                   (* Call MC_Command*)
                    instGearInPos(Master := master,
                                  Slave := axis,
                                  Enable := statBasicCommand.8 OR statFirstCycleBasicMotion,(* Input: gearInAbsolute*)
                                  GearRatio := statRatioNumerator,
                                  (*RatioDenominator :=  statRatioDenominator,*)
                                  (*MasterSyncPosition :=  statMasterSyncPosition,*)
                                  (*SlaveSyncPosition :=  statSlaveSyncPosition,*)
                                  (*SyncProfileReference :=  statSyncProfileReference,*)
                                  (*MasterStartDistance :=  statMasterStartDistance,*)

                                  Acceleration :=  statAcceleration,
                                  Deceleration :=  statDeceleration,
                                  Jerk := statJerk,
                    (*SyncDirection :=  statSyncDirection*) );


                   (* Evaluate MC_Command*)
                    IF (instGearInPos.Busy = FALSE) AND
                        (instGearInPos.Error = FALSE) AND
                        (instGearInPos.CommandAborted = FALSE) AND
                    (*( instGearInPos.StartSync = FALSE) AND*)
                        (instGearInPos.InGear = FALSE)
                        THEN
                       (* Return to NO_SELECTION if command finished*)
                        statBasicMotionState := NO_SELECTION;

                    ELSIF (instGearInPos.Error = TRUE) THEN
                       (* Errorhandling*)
                        statStatus                    := ERR_MC_GEARINPOS;
                        statErrorAutoCleared          := TRUE;
                        diagnostics                   := statDiagnostics;
                        diagnostics.subfunctionStatus := instGearInPos.ErrorId;
                        statRatioChangeOnTheFly       := FALSE;
                       (* Set next state*)
                        statFBState          := AXIS_STOP_ON_ERROR_SELECTION;
                        statBasicMotionState := NO_SELECTION;

                    ELSE
                        ;(* Command selected*)
                    END_IF;

                   (* Write MC_Command outputs to internal variable*)
                    statExeOfBasicMotion   := 16#0;
                    statExeOfBasicMotion.0 := instGearInPos.Busy;
                    statExeOfBasicMotion.2 := instGearInPos.CommandAborted;
                    statExeOfBasicMotion.3 := instGearInPos.Error;
                    (*statExeOfBasicMotion.6 :=  instGearInPos.StartSync;*)
                    (*statExeOfBasicMotion.6 :=  instGearInPos.StartSync;*)
                    statExeOfBasicMotion.7 := instGearInPos.InGear;
                {END_REGION}

                CAM_IN_SELECTED:
                   (* Additional feature (applicative): Check DB of Cam *)
                    {REGION "CAM_IN_SELECTED"}
                   (* Firstcycle of command*)
                    IF (statFirstCycleBasicMotion = TRUE) THEN
                        (*IF TypeOfDB( cam) = TO_Cam*)
                        IF tempFalse = FALSE
                            THEN
                            (*statCam :=  cam;*)
                           (* Reset CAM_IN command *)
(*                            instCamIn(Master := master,
                                      Slave := axis,
                                      (*Cam :=  statCam,*)
                                      Execute := FALSE);
*)
                            statApplicativeBasicMotionError := FALSE;
                            statApplicationMode             := configuration.camIn.applicationMode;
                        ELSE
                           (* Errorhandling - Invalid cam*)
                            statStatus                      := ERR_INVALID_CAM;
                            statErrorAutoCleared            := TRUE;
                            diagnostics.subfunctionStatus   := 0;
                            diagnostics                     := statDiagnostics;
                            statApplicativeBasicMotionError := TRUE;
                           (* Set next state*)
                            statFBState          := AXIS_STOP_ON_ERROR_SELECTION;
                            statBasicMotionState := NO_SELECTION;
                        END_IF;
                    END_IF;

                    IF (statApplicativeBasicMotionError = FALSE) THEN

                       (* Write MC Parameters*)
(*                        instCamIn.CamTableID                 := configuration.camIn.tableID;
                        instCamIn.StartMode                  := configuration.camIn.startMode;
                        instCamIn.MasterOffset               := configuration.camIn.masterOffset;
                        instCamIn.SlaveOffset                := configuration.camIn.slaveOffset;
                        instCamIn.MasterScaling              := configuration.camIn.masterScaling;
                        instCamIn.SlaveScaling               := configuration.camIn.slaveScaling;
						instCamIn.StartMode     			 := configuration.camIn.startMode;
                        instCamIn.Options.ActivationMode     := configuration.camIn.ActivationMode;
                        instCamIn.Options.ActivationPosition := configuration.camIn.ActivationPosition;
*)
                       (* Call MC_Command*)
(*                        instCamIn(Master := master,
                                  Slave := axis,
*)  //                                Execute := statBasicCommand.9 OR statFirstCycleBasicMotion);
(*
                       (* Evaluate MC_Command*)
                        IF ((instCamIn.Busy = FALSE) AND
                            (instCamIn.Error = FALSE) AND
                            (instCamIn.CommandAborted = FALSE) AND
                            (instCamIn.InSync = FALSE) AND
                        (*( instCamIn.StartSync = FALSE) AND*)
                            (statBasicCommand.9 = FALSE)
                            ) AND(* V1.0.2 Wait for one cycle EndOfProfile (--> Done) before function is finished at applicationMode ONCE*)
                            ((statApplicationMode <> APPLICATION_MODE_ONCE) OR
                            ((statApplicationMode = APPLICATION_MODE_ONCE) (*AND ( instCamIn.EndOfProfile = FALSE)*) ))
                            THEN
                           (* Return to NO_SELECTION if command finished*)
                            statBasicMotionState := NO_SELECTION;

                        ELSIF (instCamIn.Error = TRUE) THEN
                           (* Errorhandling*)
                            statStatus                    := ERR_MC_CAMIN;
                            statErrorAutoCleared          := TRUE;
                            diagnostics.subfunctionStatus := instCamIn.ErrorId;
                            diagnostics.basicMotionState  := statBasicMotionState;
                            statFBState                   := AXIS_STOP_ON_ERROR_SELECTION;
                            statBasicMotionState          := NO_SELECTION;

                        ELSE
                            ;(* Command selected*)
                        END_IF;
*)
                       (* Write MC_Command outputs to internal variable*)
                        statExeOfBasicMotion   := 16#0;
//                        statExeOfBasicMotion.0 := instCamIn.Busy;
                        IF (statApplicationMode = APPLICATION_MODE_ONCE)
                            THEN
                            ; (*statExeOfBasicMotion.1 :=  instCamIn.EndOfProfile;*)
                        END_IF;

 //                       statExeOfBasicMotion.2 := instCamIn.CommandAborted;
 //                       statExeOfBasicMotion.3 := instCamIn.Error;
                        (*statExeOfBasicMotion.6 :=  instCamIn.StartSync;*)
//                        statExeOfBasicMotion.7 := instCamIn.InSync;

                    ELSE
                        ;(* InValid cam*)
                    END_IF;
            {END_REGION}

            ELSE
               (* Errorhandling*)
                statStatus                    := ERR_UNDEFINED_BASIC_MOTION_STATE;
                statErrorUserCleared          := TRUE;
                diagnostics                   := statDiagnostics;
                diagnostics.subfunctionStatus := 0;
               (* Set errorstate*)
                statFBState := FB_ERROR;
            END_CASE;

        RESET_GEARING:
           (* Abort waiting absolute gearing / camIn job if new basic motion job is selected (configuration.generalSettings.abortWaitingSyncCmd = TRUE)*)
            instGearIn(Master := master,
                       Slave := axis,
                       Execute := TRUE,
                       RatioNumerator := 1,
                       RatioDenominator := 1);(* Lowest possible gear ratio*)

            IF (instGearIn.InGear = TRUE) OR (instGearIn.CommandAborted = TRUE)
                THEN                                           (* Relative gearing command has aborted waiting absolute gearing job*)
                statMainSelectionState    := CALL_BASIC_MOTION;(* Execute new basic motion command*)
                tempStateChangeActive     := TRUE;
                statFirstCycleBasicMotion := TRUE;

            ELSIF (instGearIn.Error = TRUE)
                THEN
                statStatus                    := ERR_MC_GEARIN;
                diagnostics.subfunctionStatus := instGearIn.ErrorId;
               (*Errorhandling*)
                statErrorAutoCleared := TRUE;
                diagnostics          := statDiagnostics;
               (*Set next state*)
                statFBState            := AXIS_STOP_ON_ERROR_SELECTION;
                statMainSelectionState := CALL_BASIC_MOTION;
                statBasicMotionState   := NO_SELECTION;

            ELSE
                ;(* Command running*)
            END_IF;

           (* Write MC_Command outputs to internal variable*)
            statExeOfBasicMotion   := 16#0;
            statExeOfBasicMotion.0 := instGearIn.Busy;
    ELSE
       (* Errorhandling*)
        statStatus                    := ERR_UNDEFINED_MAIN_SELECTION_STATE;
        statErrorUserCleared          := TRUE;
        diagnostics                   := statDiagnostics;
        diagnostics.subfunctionStatus := 0;
       (* Set errorstate*)
        statFBState := FB_ERROR;
    END_CASE;

UNTIL (tempStateChangeActive = FALSE)
END_REPEAT;

{END_REGION}


(*----------------------------------------------------------------------------------------------*)
(*Execution of homing functionality *)
(*----------------------------------------------------------------------------------------------*)


{REGION "EXECUTION_OF_PASSIVE_HOMING"}
(*Statemachine for homing functionality*)
CASE statPassiveHomingState OF
   (* Selection of extended homing mode *) 
    NO_HOMING_ACTIVE:
        ;(* Do nothing*)

    STANDARD_HOMING:
       (* No additional features*)
        {REGION "STANDARD_HOMING"}
       (* Firstcycle of command*)
        IF (statFirstCycleHoming = TRUE) THEN
           (* Reset MC_HOME command*)
            instHome(Axis := axis,
                     bCalibrationCam := homingSensor,
                     Execute := FALSE);

            IF (statBasicMotionState = ACTIVE_HOMING_SELECTED) THEN
                statBasicMotionState := NO_SELECTION;
            END_IF;
        END_IF;

       (* Call MC_Command*)
        instHome(Axis := axis,
                 bCalibrationCam := homingSensor,
                 Execute := statExtendedCommand.2,(* Input: homing*)
                 Position := configuration.homing.position,
        (*Mode :=  configuration.homing.mode*) );

       (* Evaluate MC_Command*)
        IF (instHome.Busy = FALSE) AND
            (instHome.Done = FALSE) AND
            (instHome.CommandAborted = FALSE) AND
            (instHome.Error = FALSE)
            THEN
           (* Return to NO_SELECTION if command finished*)
            statPassiveHomingState := NO_HOMING_ACTIVE;

        ELSIF (instHome.Error = TRUE) THEN
           (* Errorhandling*)
            statStatus                    := ERR_MC_HOME;
            statErrorAutoCleared          := TRUE;
            diagnostics                   := statDiagnostics;
            diagnostics.subfunctionStatus := instHome.ErrorId;
            statPassiveHomingState        := NO_HOMING_ACTIVE;
           (* Set next state*)
            statFBState := AXIS_STOP_ON_ERROR_SELECTION;
        ELSE
            ;(* Command selected*)

        END_IF;

        statExeOfHoming   := 16#0;
        statExeOfHoming.0 := instHome.Busy;
        statExeOfHoming.1 := instHome.Done;
        statExeOfHoming.2 := instHome.CommandAborted;
        statExeOfHoming.3 := instHome.Error;
{END_REGION}

ELSE
   (* Errorhandling*)
    statStatus                              := ERR_INVALID_HOMING_EXTENDED_MODE;
    statErrorAutoCleared                    := TRUE;
    diagnostics                             := statDiagnostics;
    diagnostics.subfunctionStatus           := 0;
    statDiagnostics.basicMotionState        := statBasicMotionState;
    statDiagnostics.superimposedMotionState := statSupImpMotionState;
   (* Set next state*)
    statFBState            := AXIS_STOP_ON_ERROR_SELECTION;
    statBasicMotionState   := NO_SELECTION;
    statPassiveHomingState := NO_HOMING_ACTIVE;
END_CASE;

{END_REGION}


(*----------------------------------------------------------------------------------------------*)
(*Execution of functionalities of superimposed coordinate system*)
(*----------------------------------------------------------------------------------------------*)


{REGION "EXECUTION_OF_SUPERIMPOSED_COMMANDS"}
(*Statemachine for superimposed motion commands*)
(*Write diagnostics*)

statDiagnostics.basicMotionState        := statBasicMotionState;
statDiagnostics.superimposedMotionState := statSupImpMotionState;

CASE statSupImpMotionState OF
    NO_SELECTION:
        ;(* Do nothing*)

    POS_SUPERIMPOSED_SELECTED:
       (* Additional features (applicative) : Specified direction*)
        {REGION "POS_SUPERIMPOSED_SELECTED;"}
       (* Firstcycle of command*)
        IF (statFirstCycleSupImpMotion = TRUE) THEN
           (* Configurate the direction of rotation*)
            IF ((configuration.posSuperimposed.direction = 0) AND (configuration.posSuperimposed.distance >= 0.0))(* Sign of distance is evaluated*)
                OR
                (configuration.posSuperimposed.direction = FORWARD_DIR)(* Positive direction*)
                THEN
                statSupImpMotionPosition := ABS(configuration.posSuperimposed.distance);
               (* Reset MC_MOVESUPERIMPOSED command*)
                instMoveSuperimposed(Axis := axis,
                                     Execute := FALSE);

                statApplicativeSupImpMotionError := FALSE;
            ELSIF ((configuration.posSuperimposed.direction = 0) AND (configuration.posSuperimposed.distance < 0.0))(* Sign of distance is evaluated*)
                OR
                (configuration.posSuperimposed.direction = BACKWARD_DIR)(* Negative direction *)
                THEN
                statSupImpMotionPosition := -ABS(configuration.posSuperimposed.distance);
               (* Reset MC_MOVESUPERIMPOSED command*)
                instMoveSuperimposed(Axis := axis,
                                     Execute := FALSE);

                statApplicativeSupImpMotionError := FALSE;

            ELSE
               (* Errorhandling - Invalid direction*)
                statStatus                       := ERR_INVALID_POS_SUPERIMPOSED_DIR;
                statErrorAutoCleared             := TRUE;
                diagnostics                      := statDiagnostics;
                diagnostics.subfunctionStatus    := 0;
                statApplicativeSupImpMotionError := TRUE;
               (* Set next state*)
                statFBState           := AXIS_STOP_ON_ERROR_SELECTION;
                statSupImpMotionState := NO_SELECTION;
            END_IF;
        END_IF;

        IF (statApplicativeSupImpMotionError = FALSE) THEN
           (* Call MC_Command*)
            instMoveSuperimposed(Axis := axis,
                                 Execute := statSupImpCommand.0,(* Input: posSuperimposed*)
                                 Distance := statSupImpMotionPosition,
                                 VelocityDiff := configuration.posSuperimposed.velocityDiff,
                                 Acceleration := configuration.posSuperimposed.acceleration,
                                 Deceleration := configuration.posSuperimposed.deceleration,
                                 Jerk := configuration.posSuperimposed.jerk);

           (* Evaluate MC_Command*)
            IF (instMoveSuperimposed.Busy = FALSE) AND
                (instMoveSuperimposed.Error = FALSE) AND
                (instMoveSuperimposed.Done = FALSE) AND
                (instMoveSuperimposed.CommandAborted = FALSE)
                THEN
               (* Return to NO_SELECTION if command finished*)
                statSupImpMotionState := NO_SELECTION;

            ELSIF (instMoveSuperimposed.Error = TRUE) THEN
               (* Errorhandling*)
                statStatus                    := ERR_MC_MOVESUPERIMPOSED;
                statErrorAutoCleared          := TRUE;
                diagnostics                   := statDiagnostics;
                diagnostics.subfunctionStatus := instMoveSuperimposed.ErrorId;
               (* Set next state*)
                statFBState           := AXIS_STOP_ON_ERROR_SELECTION;
                statSupImpMotionState := NO_SELECTION;

            ELSE
                ;(* command selected*)
            END_IF;

            statExeOfSupImpMotionState   := 16#0;
            statExeOfSupImpMotionState.0 := instMoveSuperimposed.Busy;
            statExeOfSupImpMotionState.1 := instMoveSuperimposed.Done;
            statExeOfSupImpMotionState.2 := instMoveSuperimposed.CommandAborted;
            statExeOfSupImpMotionState.3 := instMoveSuperimposed.Error;
        END_IF;
    {END_REGION}

    PHASING_SELECTED:
       (* Additional features (applicative) : Change setpoint on the fly (phaseShift)*)
        {REGION "PHASING_SELECTED"}
       (* Firstcycle of command*)
        IF (statFirstCycleSupImpMotion = TRUE) THEN
           (* Reset MC_PHASING_ABSOLUTE command*)
            instPhasingAbsolute(Master := master,
                                Slave := axis,
                                Execute := FALSE);

           (* Reset MC_PHASING_RELATIVE command*)
            instPhasingRelative(Master := master,
                                Slave := axis,
                                Execute := FALSE);

            statPhaseShift               := configuration.phasing.phaseShift;
            statVelocity                 := configuration.phasing.velocity;
            statAcceleration             := configuration.phasing.acceleration;
            statDeceleration             := configuration.phasing.deceleration;
            statJerk                     := configuration.phasing.jerk;
            statPhaseAbsolute            := configuration.phasing.phaseAbsolute;
            statChangePhaseShiftOnTheFly := configuration.phasing.phaseShiftChangeOnTheFly;

        ELSIF ((statChangePhaseShiftOnTheFly = TRUE) AND
            (configuration.phasing.phaseShift <> statPhaseShift)) AND
            (statPhaseAbsolute = TRUE) AND
            (instPhasingAbsolute.CommandAborted = FALSE)
            THEN
           (* Reset MC_PHASING_ABSOLUTE command - Phaseshift on the fly is only possible at phasing absolut*)
            instPhasingAbsolute(Master := master,
                                Slave := axis,
                                Execute := FALSE);

            statPhaseShift := configuration.phasing.phaseShift;
        END_IF;

       (* Select phasing absolut or relative *)
        IF (statPhaseAbsolute = TRUE) THEN
           (* Absolute phasing*)
           (* Call MC_Command*)
            instPhasingAbsolute(Master := master,
                                Slave := axis,
                                Execute := statSupImpCommand.1,(* Input: phasing*)
                                PhaseShift := statPhaseShift,
                                Velocity := statVelocity,
                                Acceleration := statAcceleration,
                                Deceleration := statDeceleration,
                                Jerk := statJerk);

           (* Evaluate MC_Command*)
            IF (instPhasingAbsolute.Busy = FALSE) AND
                (instPhasingAbsolute.Error = FALSE) AND
                (instPhasingAbsolute.Done = FALSE) AND
                (instPhasingAbsolute.CommandAborted = FALSE)
                THEN
               (* Return to NO_SELECTION if command finished*)
                statSupImpMotionState := NO_SELECTION;

            ELSIF (instPhasingAbsolute.Error = TRUE) THEN
               (* Errorhandling*)
                statStatus                    := ERR_MC_PHASINGABSOLUTE;
                statErrorAutoCleared          := TRUE;
                diagnostics                   := statDiagnostics;
                diagnostics.subfunctionStatus := instPhasingAbsolute.ErrorId;
                statChangePhaseShiftOnTheFly  := FALSE;
               (* Set next state*)
                statFBState           := AXIS_STOP_ON_ERROR_SELECTION;
                statSupImpMotionState := NO_SELECTION;

            ELSE
                ;(* Command busy*)
            END_IF;

            statExeOfSupImpMotionState   := 16#0;
            statExeOfSupImpMotionState.0 := instPhasingAbsolute.Busy;
            statExeOfSupImpMotionState.1 := instPhasingAbsolute.Done;
            statExeOfSupImpMotionState.2 := instPhasingAbsolute.CommandAborted;
            statExeOfSupImpMotionState.3 := instPhasingAbsolute.Error;

        ELSE
           (* Relative phasing  *)
           (* Call MC_Command*)
            instPhasingRelative(Master := master,
                                Slave := axis,
                                Execute := statSupImpCommand.1,(* Input: phasing*)
                                PhaseShift := statPhaseShift,
                                Velocity := statVelocity,
                                Acceleration := statAcceleration,
                                Deceleration := statDeceleration,
                                Jerk := statJerk);

           (* Evaluate MC_Command*)
            IF (instPhasingRelative.Busy = FALSE) AND
                (instPhasingRelative.Error = FALSE) AND
                (instPhasingRelative.Done = FALSE) AND
                (instPhasingRelative.CommandAborted = FALSE)
                THEN
               (* Return to NO_SELECTION if command finished*)
                statSupImpMotionState := NO_SELECTION;

            ELSIF (instPhasingRelative.Error = TRUE) THEN
               (* Errorhandling*)
                statStatus                    := ERR_MC_PHASINGRELATIVE;
                statErrorAutoCleared          := TRUE;
                diagnostics                   := statDiagnostics;
                diagnostics.subfunctionStatus := instPhasingRelative.ErrorId;
                statChangePhaseShiftOnTheFly  := FALSE;
               (* Set next state*)
                statFBState           := AXIS_STOP_ON_ERROR_SELECTION;
                statSupImpMotionState := NO_SELECTION;
            ELSE
                ;(* Command selected*)
            END_IF;

            statExeOfSupImpMotionState   := 16#0;
            statExeOfSupImpMotionState.0 := instPhasingRelative.Busy;
            statExeOfSupImpMotionState.1 := instPhasingRelative.Done;
            statExeOfSupImpMotionState.2 := instPhasingRelative.CommandAborted;
            statExeOfSupImpMotionState.3 := instPhasingRelative.Error;
        END_IF;
{END_REGION}

ELSE
   (* Errorhandling*)
    statStatus                    := ERR_UNDEFINED_SUPERIMPOSED_MOTION_STATE;
    statErrorUserCleared          := TRUE;
    diagnostics                   := statDiagnostics;
    diagnostics.subfunctionStatus := 0;
   (* Set errorstate*)
    statFBState := FB_ERROR;
END_CASE;

{END_REGION}

(*----------------------------------------------------------------------------------------------*)
(*Execution of torquelimiting functionality*)
(*----------------------------------------------------------------------------------------------*)


{REGION "EXECUTION_OF_TORQUELIMTING"}
(*Statemachine for torquelimiting *)
REPEAT
    tempStateChangeActive := FALSE;
    CASE statTorqueLimitingState OF
        NO_TORQUE_LIMITING_ACTIVE:
            ;(* Torquelimiting disable*)
       (*  instTorqueLimiting(Axis :=  axis, V01.00.03 Dont Call MC_TORQUELIMITING if disabled*)
       (*                     Enable := FALSE);*)

        TORQUE_LIMITING_DISABLE:
           (* Torquelimiting disable*)
            instTorqueLimiting(Axis := axis,
                               Enable := FALSE);

           (* Check state of torque limting*)
            IF (instTorqueLimiting.Busy = FALSE)
                THEN
               (* set next state*)
                statTorqueLimitingState := NO_TORQUE_LIMITING_ACTIVE;
            ELSE
                ;(* Waiting for MC_Torquelimiting is not busy*)
            END_IF;

        TORQUE_LIMTING_SELECTED:
           (* No extended homing function active*)
            instTorqueLimiting(Axis := axis,
                               Enable := statExtendedCommand.1,
                               TLimit := configuration.torqueLimiting.TorqueLimit,
                               Mode := configuration.torqueLimiting.mode);

            IF (instTorqueLimiting.Busy = FALSE) THEN
               (* Reset state*)
                statTorqueLimitingState := NO_TORQUE_LIMITING_ACTIVE;
            END_IF;

        (*
	        V1.00.03 Not required anymore
	       AUTOMATIC_MODE_CHANGE:
	        // In this state the torquelimiting function is operating with Mode 1 (Fixed stop detection) until inClamping = FALSE
	         instTorqueLimiting(Axis :=  axis,
	                            Enable := TRUE,
	                            Limit :=  configuration.homing.extendedModeTorqueLimit); // V01.00.03 Always use configured value
	        
	        IF ( configuration.torqueLimiting.mode =  MODE_FIXED_STOP_DETECTION)
	          OR ( instTorqueLimiting.InClamping = FALSE)
	        THEN
	          // Change state
	           statTorqueLimitingState :=  TORQUE_LIMTING_SELECTED;
	           tempStateChangeActive := TRUE;
	        ELSE
	          ; // Wait for InClamping = FALSE
	        END_IF;
	        *)

        FIXED_STOP_DETECTION_ACTIVE:
           (* Extended homing function active*)
            instTorqueLimiting(Axis := axis,
                               Enable := TRUE,
                               TLimit := configuration.homing.extendedModeTorqueLimit,(* V01.00.03 Always use configured value*)
                               Mode := MODE_FIXED_STOP_DETECTION);

            IF ((statHomingSubState = HOMING_IDLE) AND (statBasicMotionState = ACTIVE_HOMING_SELECTED))
                THEN
               (* Fixed stop process has finished - Axis is still in clamping*)
                statTorqueLimitingState := FIXED_STOP_DETECTION_FINISHED;
                tempStateChangeActive   := TRUE;

            ELSIF (statBasicMotionState <> ACTIVE_HOMING_SELECTED)
                THEN
               (* Error occurred - change state depending on inClamping*)
                IF (instTorqueLimiting.InClamping = TRUE)
                    THEN
                   (* Axis is in clamping*)
                    statTorqueLimitingState := FIXED_STOP_DETECTION_ERROR_IN_CLAMPING;
                    tempStateChangeActive   := TRUE;
                ELSE
                   (* Axis is in not clamping*)
                    statTorqueLimitingState := FIXED_STOP_DETECTION_ERROR_NOT_IN_CLAMPING;
                    tempStateChangeActive   := TRUE;
                END_IF;

            ELSE
                ;(* Fixed stop detection is running*)
            END_IF;

        FIXED_STOP_DETECTION_FINISHED:
           (* Homing on fixed stop process has finished*)
            instTorqueLimiting(Axis := axis,
                               Enable := TRUE,
                               TLimit := configuration.homing.extendedModeTorqueLimit,(* V01.00.03 Always use configured value*)
                               Mode := MODE_FIXED_STOP_DETECTION);

            IF (instTorqueLimiting.InClamping = FALSE)
                THEN
               (* InClamping = FALSE*)
                IF (statExtendedCommand.1 = TRUE)(* Torquelimiting*)
                    THEN
                    statTorqueLimitingState := TORQUE_LIMTING_SELECTED;
                ELSE
                    statTorqueLimitingState := TORQUE_LIMITING_DISABLE;
                END_IF;

                tempStateChangeActive := TRUE;
            ELSE
               (* InClamping = TRUE*)
                IF (statExtendedCommand.1 = TRUE)(* Torquelimiting*)
                    AND
                    (configuration.torqueLimiting.mode = MODE_FIXED_STOP_DETECTION)
                    THEN
                   (* Change State*)
                    statTorqueLimitingState := TORQUE_LIMTING_SELECTED;
                    tempStateChangeActive   := TRUE;
                ELSE
                    ;(* Wait for inClamping = FALSE*)
                END_IF;
            END_IF;

        FIXED_STOP_DETECTION_ERROR_IN_CLAMPING:
           (* Errorstate, torquelimiting is still active and axis not in clamping*)
            instTorqueLimiting(Axis := axis,
                               Enable := TRUE,
                               TLimit := configuration.homing.extendedModeTorqueLimit,(* V01.00.03 Always use configured value*)
                               Mode := MODE_FIXED_STOP_DETECTION);

            IF (instTorqueLimiting.InClamping = FALSE)
                THEN
               (* InClamping = FALSE -> reset torque limiting state*)
                statTorqueLimitingState := TORQUE_LIMITING_DISABLE;
               (* Torquelimiting disable*)
                tempStateChangeActive := TRUE;
            END_IF;

        FIXED_STOP_DETECTION_ERROR_NOT_IN_CLAMPING:
           (* Errorstate, torquelimiting is still active and axis in clamping*)
            instTorqueLimiting(Axis := axis,
                               Enable := TRUE,
                               TLimit := configuration.homing.extendedModeTorqueLimit,(* V01.00.03 Always use configured value*)
                               Mode := MODE_FIXED_STOP_DETECTION);

            IF (instTorqueLimiting.InClamping = TRUE)
                THEN
               (* InClamping = TRUE -> change state*)
                statTorqueLimitingState := FIXED_STOP_DETECTION_ERROR_IN_CLAMPING;
                tempStateChangeActive   := TRUE;

            ELSIF (statBasicMotionState <> NO_SELECTION) OR (statSupImpMotionState <> NO_SELECTION) OR (statPassiveHomingState <> NO_HOMING_ACTIVE)
                THEN
               (* New valid command is set -> reset error state*)
                statTorqueLimitingState := TORQUE_LIMITING_DISABLE;
                tempStateChangeActive   := TRUE;

            ELSE
                ;(* Waiting for new command or axis is getting in clamping*)
            END_IF;
    ELSE
       (* Errorhandling*)
        statStatus                          := ERR_UNDEFINED_TORQUE_LIMITING_STATE;
        statErrorUserCleared                := TRUE;
        diagnostics.basicMotionState        := statBasicMotionState;
        diagnostics.superimposedMotionState := statSupImpMotionState;
        diagnostics.subfunctionStatus       := 0;
       (* Set errorstate*)
        statFBState := FB_ERROR;
    END_CASE;
UNTIL (tempStateChangeActive = FALSE)
END_REPEAT;

(* Evaluate MC_Command*)
IF (instTorqueLimiting.Error = TRUE) AND ((statTorqueLimitingErrorOld = FALSE) OR (statStatus = STATUS_SUBSEQUENT_CALL)) THEN
   (* Errorhandling*)
    statStatus                          := ERR_MC_TORQUELIMITING;
    statErrorAutoCleared                := TRUE;
    diagnostics.basicMotionState        := statBasicMotionState;
    diagnostics.superimposedMotionState := statSupImpMotionState;
    diagnostics.subfunctionStatus       := instTorqueLimiting.ErrorId;
    statFBState                         := AXIS_STOP_ON_ERROR_SELECTION;

ELSIF (instTorqueLimiting.Error = FALSE) AND ((statTorqueLimitingErrorOld = TRUE) AND (statStatus = ERR_MC_TORQUELIMITING)) THEN
    statStatus           := STATUS_SUBSEQUENT_CALL;
    statErrorAutoCleared := FALSE;
ELSE
    ;
END_IF;

statTorqueLimitingErrorOld := instTorqueLimiting.Error;
{END_REGION}


(*----------------------------------------------------------------------------------------------*)
(* Selection of StopOnError / implementation of fastStop*)
(*----------------------------------------------------------------------------------------------*)

{REGION "STOP_ON_ERROR"}

(*Check for stopping if error occurred during execution of motion commands*)

IF (statFBState = AXIS_STOP_ON_ERROR_SELECTION)
    THEN
    statBasicMotionState   := NO_SELECTION;
    statSupImpMotionState  := NO_SELECTION;
    statPassiveHomingState := NO_HOMING_ACTIVE;

    IF (configuration.generalSettings.stopOnError = TRUE)
        THEN
       (* Read Statusword only when not already read out*)
        IF (tempStatusWord = 16#0)
            THEN
            tempStatusWord := axis.NcToPlc.StateDWord;
        END_IF;

       (* Evaluate error*)
        IF tempStatusWord.0 THEN
            ;(* Axis enabled*)
            IF (tempStatusWord.1 = TRUE) THEN
                ;(* TO Alarm present*)
                statFBState := AXIS_MOTION;
            ELSE
               (* No TO alarm present, set fastStop*)
                statBasicMotionState      := FAST_STOP_SELECTED;
                statFirstCycleBasicMotion := TRUE;
                statFBState               := AXIS_STOP_ON_ERROR_EXECUTION;
            END_IF;

        ELSE
            ;(* Axis disabled*)
            statFBState := AXIS_MOTION;
        END_IF;

    ELSE
       (* Dont StopOnError*)
        statFBState := AXIS_MOTION;
    END_IF;
END_IF;

(*Implementation of fastStop*)
IF (statBasicMotionState = FAST_STOP_SELECTED) THEN
   (* Additional feature: Load emergency stop dynamics (TO) if no valid dynamics are configured for fastStop*)
    {REGION "FASTSTOP SELECTED"}
   (* Firstcycle of command*)
    IF (statFirstCycleBasicMotion = TRUE) THEN
       (* Reset HALT command*)
        instHalt(Axis := axis,
                 Execute := FALSE);

        statFirstCycleDone := TRUE;
       (* Check dynamics for fastStop*)
       (* Load TO emergency Stop dynamics if value <=0 for deceleration is configured*)
        IF (configuration.fastStop.deceleration <= 0)(* V1.0.2 Read TO emergencyStop deceleration only IF fastStop.deceleration <= 0*)
            THEN
           (* Invalid fastStop dynamics configured - read emergency stop dynamics from TO*)
            (*statDeceleration :=  axis.DynamicDefaults.EmergencyDeceleration;*)
            statDeceleration := configuration.fastStop.deceleration;
        ELSE
           (* Valid fastStop dynamics configured*)
            statDeceleration := configuration.fastStop.deceleration;
        END_IF;

        statJerk              := configuration.fastStop.jerk;             (* V1.0.2 Use always configuration for jerk value*)
        statAbortAcceleration := configuration.fastStop.abortAcceleration;(* V1.0.2 Use always configuration*)
    END_IF;

   (* Call of MC_Command*)
    instHalt(Axis := axis,
             Execute := (statBasicCommand.0 OR statFirstCycleBasicMotion),
             Deceleration := statDeceleration,
             (*AbortAcceleration :=  statAbortAcceleration,*)
             Jerk := statJerk);

   (* Evaluate MC_Command*)
    IF (instHalt.Busy = FALSE) AND
        (instHalt.Error = FALSE) AND
        (instHalt.Done = FALSE) AND
        (instHalt.CommandAborted = FALSE)
        THEN
       (* Return to NO_SELECTION if command finished*)
        statFBState          := AXIS_MOTION;
        statBasicMotionState := NO_SELECTION;

    ELSIF (instHalt.Done = TRUE)
        THEN
        IF (statFirstCycleDone = TRUE)
            THEN
           (* Command is reset*)
            IF (instTorqueLimiting.Error = FALSE)(* V1.00.03 Dont reset error is pending*)
                THEN
               (* Reset status not if torquelimiting error is pending*)
                statStatus           := STATUS_SUBSEQUENT_CALL;
                statErrorAutoCleared := FALSE;
            END_IF;

            statFirstCycleDone := FALSE;
        END_IF;

    ELSIF (instHalt.Error = TRUE)
        THEN
       (* Errorhandling*)
        statStatus                          := ERR_MC_HALT;
        statErrorAutoCleared                := TRUE;
        diagnostics                         := statDiagnostics;
        diagnostics.basicMotionState        := statBasicMotionState;
        diagnostics.superimposedMotionState := statSupImpMotionState;
        diagnostics.subfunctionStatus       := instHalt.ErrorId;

    ELSE
        ;(* Command selected*)
    END_IF;

   (* Write MC_Command outputs to internal variable*)
    statExeOfBasicMotion   := 0;
    statExeOfBasicMotion.0 := instHalt.Busy;
    statExeOfBasicMotion.1 := instHalt.Done;
    statExeOfBasicMotion.2 := instHalt.CommandAborted;
    statExeOfBasicMotion.3 := instHalt.Error;
    {END_REGION}
END_IF;

{END_REGION}

(*----------------------------------------------------------------------------------------------*)
(*Store values and reset variables										*)
(*----------------------------------------------------------------------------------------------*)

{REGION "STORE_AND_RESET"}
(*Reset variables to determine first cycle of a new command*)
IF (statFirstCycleReset = TRUE) THEN
    statFirstCycleReset := FALSE;
END_IF;

IF (statFirstCycleHoming = TRUE) THEN
    statFirstCycleHoming := FALSE;
END_IF;

statHomingOld := tempHoming;

IF (statFirstCycleBasicMotion = TRUE) THEN
    statFirstCycleBasicMotion := FALSE;
END_IF;

statBasicCommandOld := statBasicCommand;

IF (statFirstCycleSupImpMotion = TRUE) THEN
    statFirstCycleSupImpMotion := FALSE;
END_IF;

statSupImpCommandOld := statSupImpCommand;

(*Store last values for edge detection*)
statEnableOld          := enable;
statEnableAxisOld      := enableAxis;
statExtendedCommandOld := statExtendedCommand;
statPowerErrorOld      := instPower.Error;
{END_REGION}


(*----------------------------------------------------------------------------------------------*)
(*Writing outputs													*)
(*----------------------------------------------------------------------------------------------*)

{REGION "WRITING_OF_OUTPUTS"}
(*Writing status outputs*)
resetActive := (statResetState = CMD_BUSY);

IF (statErrorUserCleared = TRUE) THEN
    ;(* Reset variables at ErrorUserCleared*)
    statBasicMotionState       := NO_SELECTION;
    statExeOfBasicMotion       := NO_SELECTION;
    statSupImpMotionState      := NO_SELECTION;
    statExeOfSupImpMotionState := NO_SELECTION;
    statExeOfHoming            := NO_SELECTION;
END_IF;

IF (instPower.Status = TRUE)
    THEN
   (* Axis enabled*)
    axisEnabled := TRUE;

ELSIF (instPower.Error = TRUE) AND (instPower.Status = FALSE)
    THEN
   (* Reset status if error occurred*)
    axisEnabled := FALSE;

ELSIF (instPower.Busy = FALSE)
    THEN
   (* Reset if MC_Power is not busy*)
    axisEnabled := FALSE;
ELSE
    ;
END_IF;

{REGION "WRITING_BASICMOTION_OUTPUTS"}
(*Writing Busy, Done and Aborted outputs for basic motion commands*)
IF (statBasicMotionState > NO_SELECTION) AND (statBasicMotionState < ACTIVE_HOMING_SELECTED)
    THEN
    commandBusy    := statExeOfBasicMotion.0;
    commandDone    := statExeOfBasicMotion.1;
    commandAborted := statExeOfBasicMotion.2;
    inVelocity     := statExeOfBasicMotion.4;
    inSync         := statExeOfBasicMotion.7;
    startSync      := statExeOfBasicMotion.6;
ELSE
    commandBusy    := FALSE;
    commandDone    := FALSE;
    commandAborted := FALSE;
    inVelocity     := FALSE;
    inSync         := FALSE;
    startSync      := FALSE;
END_IF;

(*Writing outputs up to LAxisCtrl_SpeedAxis*)
IF (statTorqueLimitingState = TORQUE_LIMTING_SELECTED)
(*OR ( statTorqueLimitingState =  AUTOMATIC_MODE_CHANGE) V1.0.3 TorqueLimtinig = TRUE, only when respective value used *)
    THEN
    torqueLimitingSelected := TRUE;
ELSE
    torqueLimitingSelected := FALSE;
END_IF;

inLimitation         := instTorqueLimiting.InLimitation;
fastStopSelected     := statBasicMotionState.0;
stopSelected         := statBasicMotionState.1;
jogSelected          := statBasicMotionState.2 OR statBasicMotionState.3;
moveVelocitySelected := statBasicMotionState.4;
(* Writing outputs up to LAxisCtrl_PosAxis*)
inClamping          := instTorqueLimiting.InClamping;
posRelativeSelected := statBasicMotionState.5;
posAbsoluteSelected := statBasicMotionState.6;
(* Writing outputs up to LAxisCtrl_SyncAxisRelGearing*)
gearInRelativeSelected := statBasicMotionState.7;
(* Writing outputs up to LAxisCtrl_SyncAxisCamming*)
gearInAbsoluteSelected := statBasicMotionState.8;
camInSelected          := statBasicMotionState.9;
inSimulation           := instSyncMotionSimulation.InSimulation;
{END_REGION}
{REGION "WRITING_HOMING_OUTPUTS"}

(* Writing Busy, Done and Aborted outputs for homing*)
IF (statPassiveHomingState = STANDARD_HOMING)
    THEN
    homingSelected       := TRUE;
    homingCommandBusy    := statExeOfHoming.0;
    homingCommandDone    := statExeOfHoming.1;
    homingCommandAborted := statExeOfHoming.2;
ELSE
    IF (statBasicMotionState = ACTIVE_HOMING_SELECTED)
        THEN
        homingSelected       := TRUE;
        homingCommandBusy    := statExeOfBasicMotion.0;
        homingCommandDone    := statExeOfBasicMotion.1;
        homingCommandAborted := statExeOfBasicMotion.2;
    ELSE
        homingSelected       := FALSE;
        homingCommandBusy    := FALSE;
        homingCommandDone    := FALSE;
        homingCommandAborted := FALSE;
    END_IF;
END_IF;

{END_REGION}
{REGION "WRITING_SUPERIMPOSED_OUTPUTS"}

(*Writing outputs for superimposed motion commands*)
IF (statSupImpMotionState <> NO_SELECTION)
    THEN
    superimposedBusy    := statExeOfSupImpMotionState.0;
    superimposedDone    := statExeOfSupImpMotionState.1;
    superimposedAborted := statExeOfSupImpMotionState.2;
ELSE
    superimposedBusy    := FALSE;
    superimposedDone    := FALSE;
    superimposedAborted := FALSE;
END_IF;

posSuperimposedSelected := statSupImpMotionState.0;
phasingSelected         := statSupImpMotionState.1;
{END_REGION}
{END_REGION}

(*----------------------------------------------------------------------------------------------*)
(*Error handling 													*)
(*----------------------------------------------------------------------------------------------*)

{REGION "ERROR_HANDLING"}
IF statErrorUserCleared THEN
    valid              := FALSE;
    busy               := TRUE;
    error              := TRUE;
    status             := statStatus;
    diagnostics.status := statStatus;

ELSIF statErrorAutoCleared THEN
    valid              := FALSE;
    busy               := TRUE;
    error              := TRUE;
    status             := statStatus;
    diagnostics.status := statStatus;

ELSE
   (* Process normal output values*)
    valid  := TRUE;
    error  := FALSE;
    status := statStatus;
END_IF;

{END_REGION}

(*Axis status function block call*)
(*instAxisStatus(stAxis := Axis.NcToPlc);*)

END_FUNCTION_BLOCK

// ---- Library/AxisControl/MC_TORQUELIMITING.TcPOU
FUNCTION_BLOCK MC_TORQUELIMITING
VAR_INPUT
	{attribute 'hide'} 
	Axis : AXIS_REF;
	Enable : BOOL;
	TLimit : LREAL;
	Mode : DINT;
END_VAR
VAR_OUTPUT
	InClamping : BOOL;
	InLimitation : BOOL;
	Busy : BOOL;
	Error : BOOL;
	ErrorId : WORD;
END_VAR
VAR
END_VAR

;

END_FUNCTION_BLOCK

// ---- Library/AxisControl/DataTypes/MC_SYNCHRONIZEDMOTIONSIMULATION.TcPOU
FUNCTION_BLOCK MC_SYNCHRONIZEDMOTIONSIMULATION

VAR_IN_OUT
	Slave	: AXIS_REF;	(* B *)
END_VAR


VAR_INPUT


	Enable : BOOL;

END_VAR
VAR_OUTPUT

	InSimulation	:BOOL;

Busy	:BOOL;

	Error	:BOOL;

ErrorId	:WORD;

END_VAR
VAR
END_VAR

;

END_FUNCTION_BLOCK

// ---- Library/Machine/Slitter/FunctionBlocks/FB_KnifeSharpening_old.TcPOU
FUNCTION_BLOCK FB_KnifeSharpening_old
VAR_INPUT

	machineRunning 				: BOOL;
	manualSharpening 			: BOOL;
	measuringWheelSensor 		: BOOL;
	knifeRunningMetersReset 		: BOOL;
	knifeEnabled 				: BOOL;
	measuringWheelDiameter 		: REAL	:= 154.2;
	sharpeningSetpoint 			: REAL	:= 100.0;
	sharpeningTime				: INT 		:= 5000;

END_VAR
VAR_OUTPUT

	sharpeningSolenoid 			: BOOL;
	knifeRunningMeters 			: INT;
	knifeRunningMetersTotal 		: DINT;


END_VAR
VAR

	measuringWheelSensorOld		: BOOL;

	instSharpeningTimeTON		: TON;
	manualSharpeningOld			: BOOL;
	knifeRunningMetersResetOld	: BOOL;

END_VAR

VAR PERSISTENT

	sensorPulseCounter1 			: DINT;	(*This variable increases every pulse of the measuring wheel and resets every time the knife is shapened*)
	sensorPulseCounter2 			: DINT;	(*This variable increases every pulse of the measuring wheel and resets manualy when the knife is replaced*)


END_VAR

VAR

END_VAR

VAR CONSTANT

	PI: REAL 					:= 3.14159265359;

END_VAR


(*==============================================================================================================================
CPNTeck - Automação industrial
(c)Copyright 2022 All Rights Reserved
_______________________________________________________________________________________________________________________________
Library: N/A 
Tested with: CX5140
Engineering: Twincat 2
Restrictions: -
Requirements: N/A
Functionality: This function block is used to sharp the knifes
Support: fabio@cpnteck.com.br
Note: Parameter comments are only available in language 'English (United States)'
_______________________________________________________________________________________________________________________________
Change log table:

Version  		| Date        			| Expert in charge  	| Changes applied
01.00.01		| 18.04.2023  		| Fabio Campion            | First released version



===============================================================================================================================*)


(*Measuring wheel pulse counter*)
IF measuringWheelSensor AND NOT measuringWheelSensorOld
AND knifeEnabled  THEN

	sensorPulseCounter1 := sensorPulseCounter1 + 1;
	sensorPulseCounter2 := sensorPulseCounter2 + 1;


END_IF

measuringWheelSensorOld := measuringWheelSensor;


(*Automatic / Manual shapening*)
IF knifeRunningMeters >= sharpeningSetpoint AND machineRunning
OR  manualSharpening AND NOT manualSharpeningOld  AND machineRunning THEN

	sensorPulseCounter1 := 0; (*Reset the measuring wheel pulse counter*)
	instSharpeningTimeTON.PT := DINT_TO_TIME(SharpeningTime); (*Set the timer setpoint*)
	instSharpeningTimeTON.IN := TRUE; (*Enable the timer*)
	sharpeningSolenoid := TRUE; (*Enable the sharpening solenoid*)

END_IF

ManualSharpeningOld := ManualSharpening;

IF instSharpeningTimeTON.Q  THEN

	sharpeningSolenoid := FALSE;
	instSharpeningTimeTON.IN := FALSE;

END_IF

IF knifeRunningMetersReset AND NOT knifeRunningMetersResetOld THEN

	sensorPulseCounter2 := 0;

END_IF

knifeRunningMetersResetOld := knifeRunningMetersReset;



(*Measuring wheel meters calculation*)
KnifeRunningMeters := TRUNC_INT((sensorPulseCounter1 * (MeasuringWheelDiameter * PI)) * 0.001);
KnifeRunningMetersTotal := TRUNC_INT((sensorPulseCounter2 * (MeasuringWheelDiameter * PI)) * 0.001);



instSharpeningTimeTON();

END_FUNCTION_BLOCK

// ---- Library/Machine/Slitter/FunctionBlocks/FB_PositionsGeneration.TcPOU
FUNCTION_BLOCK FB_PositionsGeneration
VAR_INPUT

	execute					: BOOL;	(*Execute function block*)
	machineConfig						: slitterConfig_TypeStruct;
	
END_VAR


VAR_IN_OUT

	currentOrder				: Order_TypeStruct;

END_VAR

VAR_OUTPUT

	error						: BOOL;
	done						: BOOL;
	busy						: BOOL;

END_VAR
VAR


	tempCurrentOrder				: Order_TypeStruct;

	executeOld 				: BOOL;
	firstOrderTotal 				: REAL;
	secondOrderTotal 			: REAL;
	firstKnifePosition 				: REAL;	(*First knife position*)
	topOrderIndex				: INT;		(*Top order index*)
	bottomOrderIndex			: INT;		(*Bottom order index*)
	toolPositionIndex 			: INT;		(*Tool position array index*)
	knifePositionTopIndex 			: INT ;	(*Knife position array index*)
	knifePositionBottomIndex 		: INT ;	(*Knife position array index*)
	scorerPositionTopIndex 		: INT ;	(*Knife position array index*)
	scorerPositionBottomIndex 		: INT ;	(*Knife position array index*)
	scorerPositionIndex			: INT;		(*Scorer position array index*)
	knifeEnabledIndex			: INT;		(*Knife enabled index*)
	scorerEnabledIndex			: INT;		(*Scorer enabled index*)
	knifeDistributionIndex			: INT;		(*Position distribution index*)
	scorerDistributionIndex			: INT;		(*Position distribution index*)
	toolPositionArrSize 			: INT ;	(*Tool position array size*)
	knifePositionArrSize 			: INT ;	(*Knife position array size*)
	scorerPositionArrSize 			: INT ;	(*Scorer position array size*)
	scorerExecTimes			: INT;		(*Execution times of the for loop - Used only for diagnostics*)
	toolDistributionIndex			: INT;		(*Index used to select the position and distribute to the desired toll (Knife or scorer)*)
	numberOfScorersTopOrder		: INT;		(*Number of scorers used in the top order*)
	numberOfScorersBottomOrder	: INT;		(*Number of scorers used in the bottom order*)

	toolPositionArr 				: ARRAY [1..30] OF REAL;
	knifePositionArr 				: ARRAY [1..20] OF REAL; (*Knife position*)
	scorerPositionArr 			: ARRAY [1..20] OF REAL; (*scorer position*)

	useOrder2 : BOOL;
	userOrder1 					: BOOL;
    topStep                 : INT;    // ToolPosition step for TOP (1 / 3 / 5) / Passo do TOP (1 / 3 / 5)
    bottomStep              : INT;    // ToolPosition step for BOTTOM (1 / 3 / 5) / Passo do BOTTOM (1 / 3 / 5)

    knifeOutIdx             : INT;    // Write index into knifePositionArr[] / Índice de escrita no knifePositionArr[]

	scorerMaxPositionIndex: INT;
	i: INT;
	nIndex: INT;
	nStartIdx: INT;
	scorerIdx: INT;
	topScorerIdx: INT;
	bottomScorerIdx: INT;
	knifePostionLimitIndex: INT;
	scorerPositionLimitIndex: INT;
	invertOrderSideOld: BOOL;
	scorerPositionDistributionDone: BOOL;
	base: INT;
	valid: BOOL;
	
    iKnf         : INT;
    iScr      : INT;

    nScrReq   : INT;
    startSlot : INT;
    endSlot   : INT;
    posIdx    : INT;	
    nKnfReq      : INT;
   	startKnife : INT;
	endKnife : INT;
	lbKnf: INT;
	knifeNum: INT;
	
idx : INT;	
	
	tempNextOrder: Order_TypeStruct;
	instTON_SaveSQLTimeOut: TON;
	
//    valid       : BOOL := FALSE;
    found       : BOOL := FALSE;

    startBase   : INT := 0;
    endBase     : INT := 0;

//    base        : INT := 0;
 //   i           : INT := 0;	
	
END_VAR



VAR CONSTANT
(*
	MACHINE_NUMBER_OF_KNIFES		: SINT		:= 5;	(* Number of knifes existing in the machine *)
	MACHINE_NUMBER_OF_SCORERS	: SINT	:= 8;	(* Number of scorers existing in the machine *)
*)
END_VAR


(*==============================================================================================================================
CPNTeck - Automação industrial
(c)Copyright 2022 All Rights Reserved
_______________________________________________________________________________________________________________________________
Library: N/A 
Tested with: CX5140
Engineering: Twincat 2
Restrictions: -
Requirements: N/A
Functionality: This function block is used to generate and distribute the position for the desired tools based in the operator input
Support: fabio@cpnteck.com.br
Note: Parameter comments are only available in language 'English (United States)'
_______________________________________________________________________________________________________________________________
Change log table:

Version  		| Date        			| Expert in charge  	| Changes applied
01.00.01		| 29.03.2023  		| Fabio Campion            | First released version



===============================================================================================================================*)

ACT_GenerateOrderPositions();

_invertOrders();

_bottomOrderDisplayControl();

METHOD PRIVATE _bottomOrderDisplayControl
VAR_INPUT
END_VAR
(*

	SHEET_WITH_NO_SCORER,		(* Sheet with no scoring marks*)
	SHEET_WITH_TWO_SCORER,		(* Sheet with two socoring marks *)
	SHEET_WITH_FOUR_SCORER		(*Sheet with four socoring marks*)

*)
(*
IF NOT currentOrder.secondOrderEnabled THEN
	
	currentOrder.bottom.sheetType := 0;
	currentOrder.bottom.sheetQuantity := 0;
	currentOrder.bottom.sheetM1 := 0;
	currentOrder.bottom.sheetM2 := 0;
	currentOrder.bottom.sheetM3 := 0;
	currentOrder.bottom.sheetM4 := 0;

END_IF

IF currentOrder.bottom.sheetType = SHEET_WITH_NO_SCORER THEN
	
	currentOrder.bottom.sheetM2 := 0;
	currentOrder.bottom.sheetM3 := 0;
	currentOrder.bottom.sheetM4 := 0;

END_IF

IF currentOrder.bottom.sheetType = SHEET_WITH_TWO_SCORER THEN
	
	currentOrder.bottom.sheetM4 := 0;

END_IF



IF currentOrder.top.sheetType = SHEET_WITH_NO_SCORER THEN
	
	currentOrder.top.sheetM2 := 0;
	currentOrder.top.sheetM3 := 0;
	currentOrder.top.sheetM4 := 0;

END_IF

IF currentOrder.top.sheetType = SHEET_WITH_TWO_SCORER THEN
	
	currentOrder.top.sheetM4 := 0;

END_IF
*)
END_METHOD

METHOD PRIVATE _checkOrderLimits
VAR_INPUT
END_VAR

//-------------------------------------------------------------------------------------------------
// Validate tool positions - Limits + Knife Sequence + Scorer Axis Sequence
//-------------------------------------------------------------------------------------------------
// Reset overall status flag
currentOrder.generatedOrder.statusWord.orderNotOk := FALSE;

// --- 1. KNIFE VALIDATION (Continuous Sequence: 1 < 2 < 3...) ---
FOR i := 1 TO machineConfig.machineNumberOfKnifes DO
    // Reset individual flag before checks
    currentOrder.generatedOrder.statusWord.knifeOutOfRangeArr[i] := FALSE;

    // Physical Limits
    IF currentOrder.generatedOrder.knifePositionReferenceArr[i] > machineConfig.knifeMaxPostionArr[i] OR
       currentOrder.generatedOrder.knifePositionReferenceArr[i] < machineConfig.knifeMinPostionArr[i] THEN
        currentOrder.generatedOrder.statusWord.knifeOutOfRangeArr[i] := TRUE;
        currentOrder.generatedOrder.statusWord.orderNotOk := TRUE;
    END_IF

    // Sequence Check (Next tool: i + 1)
    IF i < machineConfig.machineNumberOfKnifes THEN
        IF currentOrder.generatedOrder.knifePositionReferenceArr[i] >=
           currentOrder.generatedOrder.knifePositionReferenceArr[i + 1] THEN
            currentOrder.generatedOrder.statusWord.knifeOutOfRangeArr[i] := TRUE;
            currentOrder.generatedOrder.statusWord.knifeOutOfRangeArr[i + 1] := TRUE;
            currentOrder.generatedOrder.statusWord.orderNotOk := TRUE;
        END_IF
    END_IF
END_FOR

// --- 2. SCORER VALIDATION (Axis Sequence: 1 < 3 < 5... and 2 < 4 < 6...) ---
FOR i := 1 TO machineConfig.machineNumberOfScorers DO
    // Reset individual flag before checks
    currentOrder.generatedOrder.statusWord.scorerOutOfRangeArr[i] := FALSE;

    // Physical Limits
    IF currentOrder.generatedOrder.scorerPositionReferenceArr[i] > machineConfig.scorerMaxPostionArr[i] OR
       currentOrder.generatedOrder.scorerPositionReferenceArr[i] < machineConfig.scorerMinPostionArr[i] THEN
        currentOrder.generatedOrder.statusWord.scorerOutOfRangeArr[i] := TRUE;
        currentOrder.generatedOrder.statusWord.orderNotOk := TRUE;
    END_IF

    // Axis Sequence Check (Next tool on same axis: i + 2)
    IF (i + 2) <= machineConfig.machineNumberOfScorers THEN
        IF currentOrder.generatedOrder.scorerPositionReferenceArr[i] >=
           currentOrder.generatedOrder.scorerPositionReferenceArr[i + 2] THEN
            currentOrder.generatedOrder.statusWord.scorerOutOfRangeArr[i] := TRUE;
            currentOrder.generatedOrder.statusWord.scorerOutOfRangeArr[i + 2] := TRUE;
            currentOrder.generatedOrder.statusWord.orderNotOk := TRUE;
        END_IF
    END_IF
END_FOR
END_METHOD

METHOD PRIVATE _invertOrders
VAR_INPUT
END_VAR
// ==========================================================================
// ORDER INVERSION LOGIC (TOP/BOTTOM SWAP)
// Logic: Swaps Order 1 and Order 2 on the rising edge of the 'invert' flag
// ==========================================================================

// ---------------------------------------------------------
// CURRENT ORDER SWAP
// ---------------------------------------------------------

IF currentOrder.levelSelector =  E_LevelSelector.eBoth THEN
	
	IF currentOrder.invertOrderSide AND NOT invertOrderSideOld THEN
	
		// Backup current structure to allow safe swapping
		tempCurrentOrder := currentOrder;
	
		// Swap top and bottom orders
		currentOrder.order1 := tempCurrentOrder.order2;
		currentOrder.order2 := tempCurrentOrder.order1;
	
	END_IF
	
END_IF

// ---------------------------------------------------------
// NEXT ORDER SWAP
// ---------------------------------------------------------
IF nextOrder.levelSelector =  E_LevelSelector.eBoth THEN
	
	IF nextOrder.invertOrderSide AND NOT invertOrderSideOld THEN
	
		// Backup current structure to allow safe swapping
		tempNextOrder := nextOrder;
	
		// Swap top and bottom orders
		nextOrder.order1 := tempNextOrder.order2;
		nextOrder.order2 := tempNextOrder.order1;
	
	END_IF
		
END_IF

invertOrderSideOld := currentOrder.invertOrderSide OR nextOrder.invertOrderSide;
END_METHOD

METHOD _scorerPositionDistribution
VAR_INPUT
END_VAR
(*===============================================================================================================================
CPNTeck - Automação Industrial
(c)Copyright 2022-2025 All Rights Reserved
_______________________________________________________________________________________________________________________________
Library: N/A
Tested with: CX5140, CX9220, C6017
Engineering: TwinCAT 3
Restrictions: -
Requirements: N/A
Functionality: This function block distributes the position for the desired scorer.
Support: fabio@cpnteck.com.br
_______________________________________________________________________________________________________________________________
Change log table:
Version      | Date          | Expert in charge | Changes applied
01.00.05     | 17.02.2026    | Gemini AI        | MRBRASIL Version: Standardized to order1/order2 naming.
                                               | Kept active Home Position reset for safety.
===============================================================================================================================*)

// Verifica se ambos os pedidos não possuem vincadores
IF currentOrder.order1.sheetType = SHEET_WITH_NO_SCORER AND currentOrder.order2.sheetType = SHEET_WITH_NO_SCORER THEN
    // No scorers needed → send all tools to home and disable them
    FOR i := 1 TO 8 DO
        currentOrder.generatedOrder.scorerPositionReferenceArr[i] := machineConfig.homePositionScorer[i];
        currentOrder.generatedOrder.scorerEnabledArr[i] := FALSE;
    END_FOR

ELSE
    // Default: Reset preventivo (Garante que ferramentas não usadas voltem ao Home)
    FOR i := 1 TO 8 DO
        currentOrder.generatedOrder.scorerPositionReferenceArr[i] := machineConfig.homePositionScorer[i];
        currentOrder.generatedOrder.scorerEnabledArr[i] := FALSE;
    END_FOR

    //──────────────────────────────────────────────────────────────────────────────
    // Order 1 Logic (Equivalente ao Top)
    //──────────────────────────────────────────────────────────────────────────────
    CASE currentOrder.order1.sheetQuantity OF
        1:
            CASE currentOrder.order1.sheetType OF
                SHEET_WITH_TWO_SCORER:
                    // Option 1: Use scorers 3 and 4 if within limits
                    IF NOT (scorerPositionArr[1] > machineConfig.scorerMaxPostionArr[3] OR
                        scorerPositionArr[2] > machineConfig.scorerMaxPostionArr[4] OR
                        scorerPositionArr[1] < machineConfig.scorerMinPostionArr[3] OR
                        scorerPositionArr[2] < machineConfig.scorerMinPostionArr[4]) THEN
                        currentOrder.generatedOrder.scorerPositionReferenceArr[3] := scorerPositionArr[1];
                        currentOrder.generatedOrder.scorerPositionReferenceArr[4] := scorerPositionArr[2];
                        currentOrder.generatedOrder.scorerEnabledArr[3] := TRUE;
                        currentOrder.generatedOrder.scorerEnabledArr[4] := TRUE;
                
                    // Option 2: Try scorers 5 and 6
                    ELSIF NOT (scorerPositionArr[1] > machineConfig.scorerMaxPostionArr[5] OR
                        scorerPositionArr[2] > machineConfig.scorerMaxPostionArr[6] OR
                        scorerPositionArr[1] < machineConfig.scorerMinPostionArr[5] OR
                        scorerPositionArr[2] < machineConfig.scorerMinPostionArr[6]) THEN
                        currentOrder.generatedOrder.scorerPositionReferenceArr[5] := scorerPositionArr[1];
                        currentOrder.generatedOrder.scorerPositionReferenceArr[6] := scorerPositionArr[2];
                        currentOrder.generatedOrder.scorerEnabledArr[5] := TRUE;
                        currentOrder.generatedOrder.scorerEnabledArr[6] := TRUE;
                
                    // Option 3: Try scorers 3 and 5
                    ELSIF NOT (scorerPositionArr[1] > machineConfig.scorerMaxPostionArr[3] OR
                        scorerPositionArr[2] > machineConfig.scorerMaxPostionArr[5] OR
                        scorerPositionArr[1] < machineConfig.scorerMinPostionArr[3] OR
                        scorerPositionArr[2] < machineConfig.scorerMinPostionArr[5]) THEN
                        currentOrder.generatedOrder.scorerPositionReferenceArr[3] := scorerPositionArr[1];
                        currentOrder.generatedOrder.scorerPositionReferenceArr[5] := scorerPositionArr[2];
                        currentOrder.generatedOrder.scorerEnabledArr[3] := TRUE;
                        currentOrder.generatedOrder.scorerEnabledArr[5] := TRUE;
                
                    // Option 4: Try scorers 4 and 6
                    ELSIF NOT (scorerPositionArr[1] > machineConfig.scorerMaxPostionArr[4] OR
                        scorerPositionArr[2] > machineConfig.scorerMaxPostionArr[6] OR
                        scorerPositionArr[1] < machineConfig.scorerMinPostionArr[4] OR
                        scorerPositionArr[2] < machineConfig.scorerMinPostionArr[6]) THEN
                        currentOrder.generatedOrder.scorerPositionReferenceArr[4] := scorerPositionArr[1];
                        currentOrder.generatedOrder.scorerPositionReferenceArr[6] := scorerPositionArr[2];
                        currentOrder.generatedOrder.scorerEnabledArr[4] := TRUE;
                        currentOrder.generatedOrder.scorerEnabledArr[6] := TRUE;
                    END_IF;

                SHEET_WITH_FOUR_SCORER:
                    FOR i := 1 TO 4 DO
                        currentOrder.generatedOrder.scorerPositionReferenceArr[i] := scorerPositionArr[i];
                        currentOrder.generatedOrder.scorerEnabledArr[i] := TRUE;
                    END_FOR;
            END_CASE;

        2:
            CASE currentOrder.order1.sheetType OF
                SHEET_WITH_TWO_SCORER:
                    FOR i := 1 TO 4 DO
                        currentOrder.generatedOrder.scorerPositionReferenceArr[i] := scorerPositionArr[i];
                        currentOrder.generatedOrder.scorerEnabledArr[i] := TRUE;
                    END_FOR;
                SHEET_WITH_FOUR_SCORER:
                    FOR i := 1 TO 8 DO
                        currentOrder.generatedOrder.scorerPositionReferenceArr[i] := scorerPositionArr[i];
                        currentOrder.generatedOrder.scorerEnabledArr[i] := TRUE;
                    END_FOR;
            END_CASE;

        3:
            FOR i := 1 TO 6 DO
                currentOrder.generatedOrder.scorerPositionReferenceArr[i + 1] := scorerPositionArr[i];
                currentOrder.generatedOrder.scorerEnabledArr[i + 1] := TRUE;
            END_FOR;

        4, 5:
            FOR i := 1 TO 8 DO
                currentOrder.generatedOrder.scorerPositionReferenceArr[i] := scorerPositionArr[i];
                currentOrder.generatedOrder.scorerEnabledArr[i] := TRUE;
            END_FOR;
    END_CASE;

    //──────────────────────────────────────────────────────────────────────────────
    // Order 2 Logic (Equivalente ao Bottom)
    //──────────────────────────────────────────────────────────────────────────────
    IF currentOrder.order2.sheetQuantity > 0 THEN
        // If no order1 scorers → we can start from position 1
        IF currentOrder.order1.sheetQuantity > 0 AND currentOrder.order1.sheetType = SHEET_WITH_NO_SCORER THEN
            CASE currentOrder.order2.sheetQuantity OF
                1:
                    CASE currentOrder.order2.sheetType OF
                        SHEET_WITH_TWO_SCORER:
                            IF NOT (scorerPositionArr[1] > machineConfig.scorerMaxPostionArr[3] OR
                                scorerPositionArr[2] > machineConfig.scorerMaxPostionArr[4] OR
                                scorerPositionArr[1] < machineConfig.scorerMinPostionArr[3] OR
                                scorerPositionArr[2] < machineConfig.scorerMinPostionArr[4]) THEN
                                currentOrder.generatedOrder.scorerPositionReferenceArr[3] := scorerPositionArr[1];
                                currentOrder.generatedOrder.scorerPositionReferenceArr[4] := scorerPositionArr[2];
                                currentOrder.generatedOrder.scorerEnabledArr[3] := TRUE;
                                currentOrder.generatedOrder.scorerEnabledArr[4] := TRUE;
                            ELSIF NOT (scorerPositionArr[1] > machineConfig.scorerMaxPostionArr[5] OR
                                scorerPositionArr[2] > machineConfig.scorerMaxPostionArr[6] OR
                                scorerPositionArr[1] < machineConfig.scorerMinPostionArr[5] OR
                                scorerPositionArr[2] < machineConfig.scorerMinPostionArr[6]) THEN
                                currentOrder.generatedOrder.scorerPositionReferenceArr[5] := scorerPositionArr[1];
                                currentOrder.generatedOrder.scorerPositionReferenceArr[6] := scorerPositionArr[2];
                                currentOrder.generatedOrder.scorerEnabledArr[5] := TRUE;
                                currentOrder.generatedOrder.scorerEnabledArr[6] := TRUE;
                            END_IF;
                        SHEET_WITH_FOUR_SCORER:
                            FOR i := 1 TO 4 DO
                                currentOrder.generatedOrder.scorerPositionReferenceArr[i] := scorerPositionArr[i];
                                currentOrder.generatedOrder.scorerEnabledArr[i] := TRUE;
                            END_FOR;
                    END_CASE;

                2:
                    FOR i := 1 TO 4 DO
                        currentOrder.generatedOrder.scorerPositionReferenceArr[i + 4] := scorerPositionArr[i];
                        currentOrder.generatedOrder.scorerEnabledArr[i + 4] := TRUE;
                    END_FOR;

                3:
                    FOR i := 1 TO 6 DO
                        currentOrder.generatedOrder.scorerPositionReferenceArr[i] := scorerPositionArr[i];
                        currentOrder.generatedOrder.scorerEnabledArr[i] := TRUE;
                    END_FOR;

                4, 5:
                    FOR i := 1 TO 8 DO
                        currentOrder.generatedOrder.scorerPositionReferenceArr[i] := scorerPositionArr[i];
                        currentOrder.generatedOrder.scorerEnabledArr[i] := TRUE;
                    END_FOR;
            END_CASE;

        ELSE
            // Order 1 exists → start order 2 from scorer 5
            CASE currentOrder.order2.sheetQuantity OF
                1:
                    CASE currentOrder.order2.sheetType OF
                        SHEET_WITH_TWO_SCORER:
                            currentOrder.generatedOrder.scorerPositionReferenceArr[5] := scorerPositionArr[numberOfScorersTopOrder + 1];
                            currentOrder.generatedOrder.scorerPositionReferenceArr[6] := scorerPositionArr[numberOfScorersTopOrder + 2];
                            currentOrder.generatedOrder.scorerEnabledArr[5] := TRUE;
                            currentOrder.generatedOrder.scorerEnabledArr[6] := TRUE;
                        SHEET_WITH_FOUR_SCORER:
                            FOR i := 5 TO 8 DO
                                currentOrder.generatedOrder.scorerPositionReferenceArr[i] := scorerPositionArr[i - 4];
                                currentOrder.generatedOrder.scorerEnabledArr[i] := TRUE;
                            END_FOR;
                    END_CASE;

                2:
                    FOR i := 5 TO 8 DO
                        currentOrder.generatedOrder.scorerPositionReferenceArr[i] := scorerPositionArr[i - 4];
                        currentOrder.generatedOrder.scorerEnabledArr[i] := TRUE;
                    END_FOR;

                3:
                    FOR i := 5 TO 8 DO
                        currentOrder.generatedOrder.scorerPositionReferenceArr[i] := scorerPositionArr[i - 2];
                        currentOrder.generatedOrder.scorerEnabledArr[i] := TRUE;
                    END_FOR;

                4, 5:
                    FOR i := 5 TO 8 DO
                        currentOrder.generatedOrder.scorerPositionReferenceArr[i] := scorerPositionArr[i];
                        currentOrder.generatedOrder.scorerEnabledArr[i] := TRUE;
                    END_FOR;
            END_CASE;
        END_IF;
    END_IF;
END_IF;

// Final validation for safety limits
_checkOrderLimits();
END_METHOD

METHOD _scorerPositionDistribution_1
VAR_INPUT
END_VAR
valid := FALSE;
found := FALSE;
startBase := 0;
endBase := 0;

// -----------------------------------------------------------------------------
// Default: send all scorers to home and disable all
// -----------------------------------------------------------------------------
FOR i := 1 TO 8 DO
    currentOrder.generatedOrder.scorerPositionReferenceArr[i] := machineConfig.homePositionScorer[i];
    currentOrder.generatedOrder.scorerEnabledArr[i] := FALSE;
END_FOR

// -----------------------------------------------------------------------------
// If both sheets do not require scorers, keep all scorers at home
// -----------------------------------------------------------------------------
IF (currentOrder.order1.sheetType = SHEET_WITH_NO_SCORER) AND
   (currentOrder.order2.sheetType = SHEET_WITH_NO_SCORER) THEN
    // Nothing else to do
ELSE

    // -------------------------------------------------------------------------
    // Define possible starting windows according to required scorer quantity
    // -------------------------------------------------------------------------
    CASE currentOrder.generatedOrder.numberOfScorers OF
        2:
            startBase := 3;
            endBase := 6;

        4:
            startBase := 1;
            endBase := 5;

        6:
            startBase := 1;
            endBase := 3;

        8:
            startBase := 1;
            endBase := 1;

        ELSE
            startBase := 0;
            endBase := -1;
    END_CASE

    // -------------------------------------------------------------------------
    // Search for first valid scorer window
    // -------------------------------------------------------------------------
    IF startBase <= endBase THEN
        FOR base := startBase TO endBase DO
            valid := TRUE;

            FOR i := 0 TO currentOrder.generatedOrder.numberOfScorers - 1 DO
                IF (scorerPositionArr[i + 1] > machineConfig.scorerMaxPostionArr[base + i]) OR
                   (scorerPositionArr[i + 1] < machineConfig.scorerMinPostionArr[base + i]) THEN
                    valid := FALSE;
                    EXIT;
                END_IF
            END_FOR

            IF valid THEN
                FOR i := 0 TO currentOrder.generatedOrder.numberOfScorers - 1 DO
                    currentOrder.generatedOrder.scorerPositionReferenceArr[base + i] := scorerPositionArr[i + 1];
                    currentOrder.generatedOrder.scorerEnabledArr[base + i] := TRUE;
                END_FOR

                found := TRUE;
                EXIT;
            END_IF
        END_FOR
    END_IF

    // -------------------------------------------------------------------------
    // Flexible allocation fallback for dual-axis scorer layout
    // Odd axis : V1 V3 V5 V7
    // Even axis: V2 V4 V6 V8
    // Minimum spacing 130 mm applies only inside the same axis
    // -------------------------------------------------------------------------
    IF NOT found THEN

        IF currentOrder.generatedOrder.numberOfScorers = 6 THEN
			IF NOT found THEN
				IF (scorerPositionArr[1] >= machineConfig.scorerMinPostionArr[1]) AND
				   (scorerPositionArr[1] <= machineConfig.scorerMaxPostionArr[1]) AND
				   (scorerPositionArr[2] >= machineConfig.scorerMinPostionArr[2]) AND
				   (scorerPositionArr[2] <= machineConfig.scorerMaxPostionArr[2]) AND
				   (scorerPositionArr[3] >= machineConfig.scorerMinPostionArr[5]) AND
				   (scorerPositionArr[3] <= machineConfig.scorerMaxPostionArr[5]) AND
				   (scorerPositionArr[4] >= machineConfig.scorerMinPostionArr[6]) AND
				   (scorerPositionArr[4] <= machineConfig.scorerMaxPostionArr[6]) AND
				   (scorerPositionArr[5] >= machineConfig.scorerMinPostionArr[7]) AND
				   (scorerPositionArr[5] <= machineConfig.scorerMaxPostionArr[7]) AND
				   (scorerPositionArr[6] >= machineConfig.scorerMinPostionArr[8]) AND
				   (scorerPositionArr[6] <= machineConfig.scorerMaxPostionArr[8]) THEN
			
					currentOrder.generatedOrder.scorerPositionReferenceArr[1] := scorerPositionArr[1];
					currentOrder.generatedOrder.scorerPositionReferenceArr[2] := scorerPositionArr[2];
					currentOrder.generatedOrder.scorerPositionReferenceArr[3] := scorerPositionArr[1] + 120;	
					currentOrder.generatedOrder.scorerPositionReferenceArr[4] := scorerPositionArr[2] + 120;				
					currentOrder.generatedOrder.scorerPositionReferenceArr[5] := scorerPositionArr[3];
					currentOrder.generatedOrder.scorerPositionReferenceArr[6] := scorerPositionArr[4];
					currentOrder.generatedOrder.scorerPositionReferenceArr[7] := scorerPositionArr[5];
					currentOrder.generatedOrder.scorerPositionReferenceArr[8] := scorerPositionArr[6];
			
					currentOrder.generatedOrder.scorerEnabledArr[1] := TRUE;
					currentOrder.generatedOrder.scorerEnabledArr[2] := TRUE;
					currentOrder.generatedOrder.scorerEnabledArr[5] := TRUE;
					currentOrder.generatedOrder.scorerEnabledArr[6] := TRUE;
					currentOrder.generatedOrder.scorerEnabledArr[7] := TRUE;
					currentOrder.generatedOrder.scorerEnabledArr[8] := TRUE;
			
					found := TRUE;
				END_IF
			END_IF		
		
				
		
            // -----------------------------------------------------------------
            // Pattern: V1 V2 V3 V4 V5 V7
            // -----------------------------------------------------------------
			IF NOT found THEN
				IF (scorerPositionArr[1] >= machineConfig.scorerMinPostionArr[1]) AND
				   (scorerPositionArr[1] <= machineConfig.scorerMaxPostionArr[1]) AND
				   (scorerPositionArr[2] >= machineConfig.scorerMinPostionArr[2]) AND
				   (scorerPositionArr[2] <= machineConfig.scorerMaxPostionArr[2]) AND
				   (scorerPositionArr[3] >= machineConfig.scorerMinPostionArr[3]) AND
				   (scorerPositionArr[3] <= machineConfig.scorerMaxPostionArr[3]) AND
				   (scorerPositionArr[4] >= machineConfig.scorerMinPostionArr[4]) AND
				   (scorerPositionArr[4] <= machineConfig.scorerMaxPostionArr[4]) AND
				   (scorerPositionArr[5] >= machineConfig.scorerMinPostionArr[5]) AND
				   (scorerPositionArr[5] <= machineConfig.scorerMaxPostionArr[5]) AND
				   (scorerPositionArr[6] >= machineConfig.scorerMinPostionArr[7]) AND
				   (scorerPositionArr[6] <= machineConfig.scorerMaxPostionArr[7]) THEN
	
					currentOrder.generatedOrder.scorerPositionReferenceArr[1] := scorerPositionArr[1];
					currentOrder.generatedOrder.scorerPositionReferenceArr[2] := scorerPositionArr[2];
					currentOrder.generatedOrder.scorerPositionReferenceArr[3] := scorerPositionArr[3];
					currentOrder.generatedOrder.scorerPositionReferenceArr[4] := scorerPositionArr[4];
					currentOrder.generatedOrder.scorerPositionReferenceArr[5] := scorerPositionArr[5];
					currentOrder.generatedOrder.scorerPositionReferenceArr[7] := scorerPositionArr[6];
	
					currentOrder.generatedOrder.scorerEnabledArr[1] := TRUE;
					currentOrder.generatedOrder.scorerEnabledArr[2] := TRUE;
					currentOrder.generatedOrder.scorerEnabledArr[3] := TRUE;
					currentOrder.generatedOrder.scorerEnabledArr[4] := TRUE;
					currentOrder.generatedOrder.scorerEnabledArr[5] := TRUE;
					currentOrder.generatedOrder.scorerEnabledArr[7] := TRUE;
	
					found := TRUE;
				END_IF
            END_IF

            // -----------------------------------------------------------------
            // Pattern: V2 V3 V4 V5 V7 V8
            // -----------------------------------------------------------------
            IF NOT found THEN
                IF (scorerPositionArr[1] >= machineConfig.scorerMinPostionArr[2]) AND
                   (scorerPositionArr[1] <= machineConfig.scorerMaxPostionArr[2]) AND
                   (scorerPositionArr[2] >= machineConfig.scorerMinPostionArr[3]) AND
                   (scorerPositionArr[2] <= machineConfig.scorerMaxPostionArr[3]) AND
                   (scorerPositionArr[3] >= machineConfig.scorerMinPostionArr[4]) AND
                   (scorerPositionArr[3] <= machineConfig.scorerMaxPostionArr[4]) AND
                   (scorerPositionArr[4] >= machineConfig.scorerMinPostionArr[5]) AND
                   (scorerPositionArr[4] <= machineConfig.scorerMaxPostionArr[5]) AND
                   (scorerPositionArr[5] >= machineConfig.scorerMinPostionArr[7]) AND
                   (scorerPositionArr[5] <= machineConfig.scorerMaxPostionArr[7]) AND
                   (scorerPositionArr[6] >= machineConfig.scorerMinPostionArr[8]) AND
                   (scorerPositionArr[6] <= machineConfig.scorerMaxPostionArr[8]) THEN

                    currentOrder.generatedOrder.scorerPositionReferenceArr[2] := scorerPositionArr[1];
                    currentOrder.generatedOrder.scorerPositionReferenceArr[3] := scorerPositionArr[2];
                    currentOrder.generatedOrder.scorerPositionReferenceArr[4] := scorerPositionArr[3];
                    currentOrder.generatedOrder.scorerPositionReferenceArr[5] := scorerPositionArr[4];
                    currentOrder.generatedOrder.scorerPositionReferenceArr[7] := scorerPositionArr[5];
                    currentOrder.generatedOrder.scorerPositionReferenceArr[8] := scorerPositionArr[6];

                    currentOrder.generatedOrder.scorerEnabledArr[2] := TRUE;
                    currentOrder.generatedOrder.scorerEnabledArr[3] := TRUE;
                    currentOrder.generatedOrder.scorerEnabledArr[4] := TRUE;
                    currentOrder.generatedOrder.scorerEnabledArr[5] := TRUE;
                    currentOrder.generatedOrder.scorerEnabledArr[7] := TRUE;
                    currentOrder.generatedOrder.scorerEnabledArr[8] := TRUE;

                    found := TRUE;
                END_IF
            END_IF

            // -----------------------------------------------------------------
            // Pattern: V1 V2 V3 V4 V6 V8
            // -----------------------------------------------------------------
            IF NOT found THEN
                IF (scorerPositionArr[1] >= machineConfig.scorerMinPostionArr[1]) AND
                   (scorerPositionArr[1] <= machineConfig.scorerMaxPostionArr[1]) AND
                   (scorerPositionArr[2] >= machineConfig.scorerMinPostionArr[2]) AND
                   (scorerPositionArr[2] <= machineConfig.scorerMaxPostionArr[2]) AND
                   (scorerPositionArr[3] >= machineConfig.scorerMinPostionArr[3]) AND
                   (scorerPositionArr[3] <= machineConfig.scorerMaxPostionArr[3]) AND
                   (scorerPositionArr[4] >= machineConfig.scorerMinPostionArr[4]) AND
                   (scorerPositionArr[4] <= machineConfig.scorerMaxPostionArr[4]) AND
                   (scorerPositionArr[5] >= machineConfig.scorerMinPostionArr[6]) AND
                   (scorerPositionArr[5] <= machineConfig.scorerMaxPostionArr[6]) AND
                   (scorerPositionArr[6] >= machineConfig.scorerMinPostionArr[8]) AND
                   (scorerPositionArr[6] <= machineConfig.scorerMaxPostionArr[8]) THEN

                    currentOrder.generatedOrder.scorerPositionReferenceArr[1] := scorerPositionArr[1];
                    currentOrder.generatedOrder.scorerPositionReferenceArr[2] := scorerPositionArr[2];
                    currentOrder.generatedOrder.scorerPositionReferenceArr[3] := scorerPositionArr[3];
                    currentOrder.generatedOrder.scorerPositionReferenceArr[4] := scorerPositionArr[4];
                    currentOrder.generatedOrder.scorerPositionReferenceArr[6] := scorerPositionArr[5];
                    currentOrder.generatedOrder.scorerPositionReferenceArr[8] := scorerPositionArr[6];

                    currentOrder.generatedOrder.scorerEnabledArr[1] := TRUE;
                    currentOrder.generatedOrder.scorerEnabledArr[2] := TRUE;
                    currentOrder.generatedOrder.scorerEnabledArr[3] := TRUE;
                    currentOrder.generatedOrder.scorerEnabledArr[4] := TRUE;
                    currentOrder.generatedOrder.scorerEnabledArr[6] := TRUE;
                    currentOrder.generatedOrder.scorerEnabledArr[8] := TRUE;

                    found := TRUE;
                END_IF
            END_IF

        END_IF
    END_IF
END_IF

// Final safety validation
_checkOrderLimits();
END_METHOD

METHOD _scorerPositionDistribution_bak
VAR_INPUT
END_VAR
(*===============================================================================================================================
CPNTeck - Automação Industrial
(c)Copyright 2022-2026 All Rights Reserved
_______________________________________________________________________________________________________________________________
Library: N/A
Tested with: CX5140, CX9220, C6017
Engineering: TwinCAT 3
Restrictions: -
Requirements: N/A
Functionality: This function block distributes the position for the desired scorer.
Support: fabio@cpnteck.com.br
_______________________________________________________________________________________________________________________________
Change log table:
Version      | Date          | Expert in charge | Changes applied
01.00.06     | 17.02.2026    | Gemini AI        | Syntax fix for TwinCAT 3 (IEC 61131-3).
                                               | Standardized to order1/order2 logic.
===============================================================================================================================*)
(*
// 1) Verificação de ausência de vincadores em ambos os pedidos
IF currentOrder.order1.sheetType = SHEET_WITH_NO_SCORER AND currentOrder.order2.sheetType = SHEET_WITH_NO_SCORER THEN
    FOR i := 1 TO 8 DO
        currentOrder.generatedOrder.scorerPositionReferenceArr[i] := machineConfig.homePositionScorer[i];
        currentOrder.generatedOrder.scorerEnabledArr[i] := FALSE;
    END_FOR
ELSE
    // Default: Reset preventivo para Home e desabilitar
    FOR i := 1 TO 8 DO
        currentOrder.generatedOrder.scorerPositionReferenceArr[i] := machineConfig.homePositionScorer[i];
        currentOrder.generatedOrder.scorerEnabledArr[i] := FALSE;
    END_FOR

    // 2) Distribuição baseada na quantidade total de vincadores gerados
    CASE currentOrder.generatedOrder.numberOfScorers OF

        2:
            (* Tenta pares em múltiplas posições *)
            FOR base := 3 TO 6 DO
                IF NOT (
                    scorerPositionArr[1] > machineConfig.scorerMaxPostionArr[base] OR
                    scorerPositionArr[2] > machineConfig.scorerMaxPostionArr[base + 1] OR
                    scorerPositionArr[1] < machineConfig.scorerMinPostionArr[base] OR
                    scorerPositionArr[2] < machineConfig.scorerMinPostionArr[base + 1]
                ) THEN
                    currentOrder.generatedOrder.scorerPositionReferenceArr[base] := scorerPositionArr[1];
                    currentOrder.generatedOrder.scorerPositionReferenceArr[base + 1] := scorerPositionArr[2];
                    currentOrder.generatedOrder.scorerEnabledArr[base] := TRUE;
                    currentOrder.generatedOrder.scorerEnabledArr[base + 1] := TRUE;
                    EXIT; 
                END_IF
            END_FOR

        4:
            (* Tenta grupos de 4 vincadores *)
            FOR base := 1 TO 5 DO
                IF NOT (
                    scorerPositionArr[1] > machineConfig.scorerMaxPostionArr[base] OR
                    scorerPositionArr[2] > machineConfig.scorerMaxPostionArr[base + 1] OR
                    scorerPositionArr[3] > machineConfig.scorerMaxPostionArr[base + 2] OR
                    scorerPositionArr[4] > machineConfig.scorerMaxPostionArr[base + 3] OR
                    scorerPositionArr[1] < machineConfig.scorerMinPostionArr[base] OR
                    scorerPositionArr[2] < machineConfig.scorerMinPostionArr[base + 1] OR
                    scorerPositionArr[3] < machineConfig.scorerMinPostionArr[base + 2] OR
                    scorerPositionArr[4] < machineConfig.scorerMinPostionArr[base + 3]
                ) THEN
                    FOR i := 0 TO 3 DO
                        currentOrder.generatedOrder.scorerPositionReferenceArr[base + i] := scorerPositionArr[i + 1];
                        currentOrder.generatedOrder.scorerEnabledArr[base + i] := TRUE;
                    END_FOR
                    EXIT;
                END_IF
            END_FOR

        6:
            (* Tenta grupos de 6 vincadores *)
            FOR base := 1 TO 3 DO
                valid := TRUE;
                FOR i := 0 TO 5 DO
                    IF scorerPositionArr[i + 1] > machineConfig.scorerMaxPostionArr[base + i] OR
                       scorerPositionArr[i + 1] < machineConfig.scorerMinPostionArr[base + i] THEN
                        valid := FALSE;
                        EXIT;
                    END_IF
                END_FOR
                
                IF valid THEN
                    FOR i := 0 TO 5 DO
                        currentOrder.generatedOrder.scorerPositionReferenceArr[base + i] := scorerPositionArr[i + 1];
                        currentOrder.generatedOrder.scorerEnabledArr[base + i] := TRUE;
                    END_FOR
                    EXIT;
                END_IF
            END_FOR

        8:
            (* Validação direta para todos os 8 vincadores *)
            valid := TRUE;
            FOR i := 1 TO 8 DO
                IF scorerPositionArr[i] > machineConfig.scorerMaxPostionArr[i] OR
                   scorerPositionArr[i] < machineConfig.scorerMinPostionArr[i] THEN
                    valid := FALSE;
                    EXIT;
                END_IF
            END_FOR
            
            IF valid THEN
                FOR i := 1 TO 8 DO
                    currentOrder.generatedOrder.scorerPositionReferenceArr[i] := scorerPositionArr[i];
                    currentOrder.generatedOrder.scorerEnabledArr[i] := TRUE;
                END_FOR
            END_IF

    END_CASE
END_IF

// 3) Validação final de segurança
_checkOrderLimits();

*)


(*===============================================================================================================================
CPNTeck - Automação Industrial
(c)Copyright 2022-2025 All Rights Reserved
_______________________________________________________________________________________________________________________________
Library: N/A
Tested with: CX5140, CX9220, C6017
Engineering: TwinCAT 3
Restrictions: -
Requirements: N/A
Functionality: This function block distributes the position for the desired scorer.
Support: fabio@cpnteck.com.br
Note: Parameter comments are only available in language 'English (United States)'
_______________________________________________________________________________________________________________________________
Change log table:
Version      | Date         | Expert in charge | Changes applied
01.00.01     | 29.03.2023   | Fabio Campion    | First released version
01.00.02     | 27.04.2025   | Fabio Campion    | Added scorerEnabledArr logic
01.00.03     | 29.04.2025   | Fabio Campion    | Fixed bottom scorer distribution if top is empty
01.00.04     | 29.04.2025   | Fabio Campion    | Unified CASE logic for bottom scorers, added collision check
01.00.05     | 28.05.2025   | Fabio Campion    | Completed logic up to 8 scorers with validation combinations
===============================================================================================================================*)

IF currentOrder.order1.sheetType = SHEET_WITH_NO_SCORER AND currentOrder.order2.sheetType = SHEET_WITH_NO_SCORER THEN
    FOR i := 1 TO 8 DO
        currentOrder.generatedOrder.scorerPositionReferenceArr[i] := machineConfig.homePositionScorer[i];
        currentOrder.generatedOrder.scorerEnabledArr[i] := FALSE;
    END_FOR
ELSE
    FOR i := 1 TO 8 DO
        currentOrder.generatedOrder.scorerPositionReferenceArr[i] := machineConfig.homePositionScorer[i];
        currentOrder.generatedOrder.scorerEnabledArr[i] := FALSE;
    END_FOR

    CASE currentOrder.generatedOrder.numberOfScorers OF

        2:
            (* Try pairs in multiple positions *)
            FOR base := 3 TO 6 BY 1 DO
                IF NOT (
                    scorerPositionArr[1] > machineConfig.scorerMaxPostionArr[base] OR
                    scorerPositionArr[2] > machineConfig.scorerMaxPostionArr[base + 1] OR
                    scorerPositionArr[1] < machineConfig.scorerMinPostionArr[base] OR
                    scorerPositionArr[2] < machineConfig.scorerMinPostionArr[base + 1]
                ) THEN
                    currentOrder.generatedOrder.scorerPositionReferenceArr[base] := scorerPositionArr[1];
                    currentOrder.generatedOrder.scorerPositionReferenceArr[base + 1] := scorerPositionArr[2];
                    currentOrder.generatedOrder.scorerEnabledArr[base] := TRUE;
                    currentOrder.generatedOrder.scorerEnabledArr[base + 1] := TRUE;
                    EXIT;
                END_IF
            END_FOR

        4:
            FOR base := 1 TO 5 BY 1 DO
                IF NOT (
                    scorerPositionArr[1] > machineConfig.scorerMaxPostionArr[base] OR
                    scorerPositionArr[2] > machineConfig.scorerMaxPostionArr[base + 1] OR
                    scorerPositionArr[3] > machineConfig.scorerMaxPostionArr[base + 2] OR
                    scorerPositionArr[4] > machineConfig.scorerMaxPostionArr[base + 3] OR
                    scorerPositionArr[1] < machineConfig.scorerMinPostionArr[base] OR
                    scorerPositionArr[2] < machineConfig.scorerMinPostionArr[base + 1] OR
                    scorerPositionArr[3] < machineConfig.scorerMinPostionArr[base + 2] OR
                    scorerPositionArr[4] < machineConfig.scorerMinPostionArr[base + 3]
                ) THEN
                    FOR i := 0 TO 3 DO
                        currentOrder.generatedOrder.scorerPositionReferenceArr[base + i] := scorerPositionArr[i + 1];
                        currentOrder.generatedOrder.scorerEnabledArr[base + i] := TRUE;
                    END_FOR
                    EXIT;
                END_IF
            END_FOR

        6:
            FOR base := 1 TO 3 BY 1 DO
                valid := TRUE;
                FOR i := 0 TO 5 DO
                    IF scorerPositionArr[i + 1] > machineConfig.scorerMaxPostionArr[base + i] OR
                       scorerPositionArr[i + 1] < machineConfig.scorerMinPostionArr[base + i] THEN
                        valid := FALSE;
                        EXIT;
                    END_IF
                END_FOR
                IF valid THEN
                    FOR i := 0 TO 5 DO
                        currentOrder.generatedOrder.scorerPositionReferenceArr[base + i] := scorerPositionArr[i + 1];
                        currentOrder.generatedOrder.scorerEnabledArr[base + i] := TRUE;
                    END_FOR
                    EXIT;
                END_IF
            END_FOR

        8:
            valid := TRUE;
            FOR i := 1 TO 8 DO
                IF scorerPositionArr[i] > machineConfig.scorerMaxPostionArr[i] OR
                   scorerPositionArr[i] < machineConfig.scorerMinPostionArr[i] THEN
                    valid := FALSE;
                    EXIT;
                END_IF
            END_FOR
            IF valid THEN
                FOR i := 1 TO 8 DO
                    currentOrder.generatedOrder.scorerPositionReferenceArr[i] := scorerPositionArr[i];
                    currentOrder.generatedOrder.scorerEnabledArr[i] := TRUE;
                END_FOR
            END_IF

    END_CASE
END_IF;

// Final safety validation
_checkOrderLimits();
END_METHOD

ACTION ACT_CalculateNumberOfKnifes:

(*==============================================================================================================================
CPNTeck - Automação industrial
(c)Copyright 2022 All Rights Reserved
_______________________________________________________________________________________________________________________________
Library: N/A 
Tested with: CX5140
Engineering: Twincat 2
Restrictions: -
Requirements: N/A
Functionality: This method is used to calculate the number of knifes used in the order entered by the operator
Support: fabio@cpnteck.com.br
Note: Parameter comments are only available in language 'English (United States)'
_______________________________________________________________________________________________________________________________
Change log table:

Version  		| Date        			| Expert in charge  	| Changes applied
01.00.01		| 29.03.2023  		| Fabio Campion            | First released version



===============================================================================================================================*)


(*Calculate the number of knifes to be used in the production*)
currentOrder.generatedOrder.numberOfKnifes := currentOrder.generatedOrder.numberOfSheets + 1;
END_ACTION

ACTION ACT_CalculateNumberOfScorers:
(*==============================================================================================================================
CPNTeck - Automação industrial
(c)Copyright 2022 All Rights Reserved
_______________________________________________________________________________________________________________________________
Library: N/A
Tested with: CX5140
Engineering: TwinCAT 2
Restrictions: -
Requirements: N/A
Functionality:
    Calculates the number of scorers required for the operator-entered order, considering the level enable mode:
      - eUpperOnly: calculate only TOP (upper) sheet
      - eLowerOnly: calculate only BOTTOM (lower) sheet
      - eBoth:      calculate TOP + BOTTOM
Support: fabio@cpnteck.com.br
Note: Parameter comments are only available in language 'English (United States)'
_______________________________________________________________________________________________________________________________
Change log table:

Version   | Date       | Expert in charge | Changes applied
01.00.01  | 29.03.2023 | Fabio Campion    | First released version
01.00.02  | 30.12.2025 | Fabio Campion    | Add E_ScorerEnableMode selection (upper/lower/both)
===============================================================================================================================*)

currentOrder.generatedOrder.numberOfScorers := 0; // Reset before calculation

// Default to zero every scan
numberOfScorersTopOrder    := 0;
numberOfScorersBottomOrder := 0;

//-------------------------------------------------------------------------------------------------
// TOP (Upper) calculation
//-------------------------------------------------------------------------------------------------
IF (currentOrder.levelSelector = E_LevelSelector.eUpperOnly)
 OR (currentOrder.levelSelector = E_LevelSelector.eLowerOnly)	
   OR (currentOrder.levelSelector = E_LevelSelector.eBoth) THEN

    CASE currentOrder.order1.sheetType OF
        SHEET_WITH_NO_SCORER:
            numberOfScorersTopOrder := 0;

        SHEET_WITH_TWO_SCORER:
            numberOfScorersTopOrder := (2 * currentOrder.order1.sheetQuantity);

        SHEET_WITH_FOUR_SCORER:
            numberOfScorersTopOrder := (4 * currentOrder.order1.sheetQuantity);
    END_CASE

END_IF

//-------------------------------------------------------------------------------------------------
// BOTTOM (Lower) calculation
//-------------------------------------------------------------------------------------------------
IF (currentOrder.levelSelector = E_LevelSelector.eBoth) THEN
	
    CASE currentOrder.order2.sheetType OF
        SHEET_WITH_NO_SCORER:
            numberOfScorersBottomOrder := 0;

        SHEET_WITH_TWO_SCORER:
            numberOfScorersBottomOrder := (2 * currentOrder.order2.sheetQuantity);

        SHEET_WITH_FOUR_SCORER:
            numberOfScorersBottomOrder := (4 * currentOrder.order2.sheetQuantity);
    END_CASE

END_IF

//-------------------------------------------------------------------------------------------------
// Total
//-------------------------------------------------------------------------------------------------
currentOrder.generatedOrder.numberOfScorers := numberOfScorersTopOrder + numberOfScorersBottomOrder;
END_ACTION

ACTION ACT_CalculateNumberOfSheets:
(*==============================================================================================================================
CPNTeck - Automação industrial
(c)Copyright 2022 All Rights Reserved
_______________________________________________________________________________________________________________________________
Library: N/A
Tested with: CX5140
Engineering: TwinCAT 2
Restrictions: -
Requirements: N/A
Functionality: This method is used to calculate the number of sheets used in the order entered by the operator,
               considering E_LevelSelector (eUpperOnly / eLowerOnly / eBoth).
Support: fabio@cpnteck.com.br
Note: Parameter comments are only available in language 'English (United States)'
_______________________________________________________________________________________________________________________________
Change log table:

Version   | Date       | Expert in charge | Changes applied
01.00.01  | 29.03.2023 | Fabio Campion    | First released version
01.00.02  | 30.12.2025 | Fabio Campion    | Add E_LevelSelector selection (upper/lower/both)
===============================================================================================================================*)

(* Calculate the number of sheets of production list *)

// Default
currentOrder.generatedOrder.numberOfSheets := 0;

CASE currentOrder.levelSelector OF

    E_LevelSelector.eUpperOnly:
        currentOrder.generatedOrder.numberOfSheets := currentOrder.order1.sheetQuantity;

    E_LevelSelector.eLowerOnly:
        currentOrder.generatedOrder.numberOfSheets := currentOrder.order1.sheetQuantity;

